SUBAPPLICATION Uebung_079 (* alle TECU FBs *)
  (* Standard: 61499-2 *)
  (* Version 1.0, 2023-10-23, franz *)
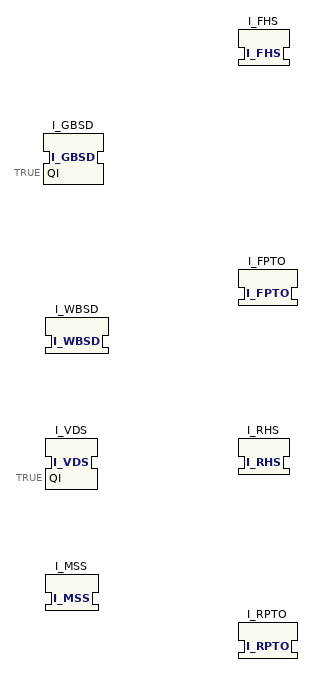
  FBS
    I_GBSD : I_GBSD(QI := TRUE);
    I_VDS : I_VDS(QI := TRUE);
    I_WBSD : I_WBSD;
    I_MSS : I_MSS;
    I_FHS : I_FHS;
    I_FPTO : I_FPTO;
    I_RHS : I_RHS;
    I_RPTO : I_RPTO;
  END_FBS
END_SUBAPPLICATION
